FUNCTION_BLOCK LPF1
VAR_INPUT
	T		: LREAL;		// Filter parameter: time constant
	K		: LREAL;		// Filter parameter: gain
	ts		: LREAL;		// Sampling time
	u		: LREAL;		// Filter input signal
END_VAR	
VAR_OUTPUT
	y		: LREAL;		// Filter output signal
END_VAR
VAR
	yLast	: LREAL := 0;	// Store last output value
END_VAR

y := yLast + (K * u - yLast) * ts / T;
yLast := y;

END_FUNCTION_BLOCK

(* stored: Version 1.1.0.1, ProductVersion 3.1.4024.11
   POU LPF1: Id {7763ceb7-d931-429f-8950-f9278aeb47f5}, SpecialFunc None *)
